// TIA Portal V20 export
// export: Created 2025-12-01T14:57:15.1286003Z, ExportSetting None, DisplayName Totally Integrated Automation Portal, DisplayVersion V20 Update 3, DisplayName TIA Portal Openness, DisplayVersion V20 Update 3, DisplayName TIA Portal Version Control Interface, DisplayVersion V20 Update 3, DisplayName STEP 7 Professional, DisplayVersion V20 Update 3, DisplayName STEP 7 Safety, DisplayVersion V20 Update 2, DisplayName WinCC Basic/Comfort/Advanced, DisplayVersion V20 Update 3, DisplayName WinCC Professional, DisplayVersion V20 Update 3, DisplayName WinCC Unified, DisplayVersion V20 Update 3
FUNCTION_BLOCK "FB900_CONTROL_ZONA"   // FB900, LAD
{ S7_Optimized_Access := 'FALSE' }
AUTHOR : ESTANDAR
NAME : 20160526
VERSION : 3.4
// stored: AutoNumber false, SetENOAutomatically false
   VAR_INPUT
      NumZonaUP : UInt;
      NumZona : UInt;
      MAR_FinReset_DW : Bool;   // FIN RESET MESAS INTEGRANTES CBOX
      CONF_Reset_Manual : Bool;   // Reset Manual
      INP_Sel_OffLine : Bool;
      INP_Sel_Main : Bool;
      INP_Pul_Marcha : Bool;   // Pulsador Manual Zona
      INP_Pul_Paro : Bool;   // Pulsador Paro Zona
      INP_Pul_Rearme : Bool;   // Pulsador Test Luces CCPIF
      INP_Pul_TLuces : Bool;   // Pulsador Test Luces Zona
      INP_Sel_Automat : Bool;   // Selector Automatico Zona
      INP_Sel_Manual : Bool;   // Selector Automatico Zona
   END_VAR
   VAR_OUTPUT
      L_Verde : Bool;   // Piloto Marcha
      L_Rojo : Bool;   // Piloto Error
      L_Naranja : Bool;
      Sirena : Bool;
   END_VAR
   VAR
      Toff_Rearme { ExternalAccessible := 'False'; ExternalVisible := 'False'; ExternalWritable := 'False'} : TOF_TIME;
      TIM_RetardoMarcha { S7_SetPoint := 'True'} : TON_TIME;
      Valor_Cuenta_Reset : UDInt;   // No comment
      Modo_Zona_E0 : Bool;   // Gragcet Modo
      Modo_Zona_E1 : Bool;   // Gragcet Modo
      Modo_Zona_E2 : Bool;   // Gragcet Modo
      Modo_Zona_E3 : Bool;   // Gragcet Modo
      Modo_Zona_E4 : Bool;   // Gragcet Modo
      Modo_Zona_E5 : Bool;   // Gragcet Modo
      S_Paro_Zona : Bool;   // Sel_Paro
      S_Marcha_Zona : Bool;   // Sel_Marcha
      Auto_Zona_E0 : Bool;   // Grafcet Auto
      Auto_Zona_E1 : Bool;   // Grafcet Auto
      Auto_Zona_E2 : Bool;   // Grafcet Auto
      Auto_Zona_E3 : Bool;   // Grafcet Auto
      Auto_Zona_E4 : Bool;   // Grafcet Auto
      Auto_Zona_E5 : Bool;   // Grafcet Auto
      Reset_Zona_E0 : Bool;   // Grafcet Reset
      Reset_Zona_E1 : Bool;   // Grafcet Reset
      Reset_Zona_E2 : Bool;   // Grafcet Reset
      Reset_Zona_E3 : Bool;   // Grafcet Reset
      Reset_Zona_E4 : Bool;   // Grafcet Reset
      Reset_Zona_E5 : Bool;   // Grafcet Reset
      Reset_Zona_E6 : Bool;   // Grafcet Reset
      Reset_Zona_E7 : Bool;   // Grafcet Reset
      Mem_PulMarcha_Zona : Bool;   // Mem_Auxiliar
      Mem_Error_Zona : Bool;   // Mem_Auxiliar
      Mem_Aviso_Error_Zona : Bool;   // Mem_Auxiliar
      Mem_Parar_Zona : Bool;   // Mem_Auxiliar
      Mem_Reseteo_Zona : Bool;   // Mem_Auxiliar
      Mem_PulParo_Zona : Bool;   // Mem_Auxiliar
      Mem_Fin_Zona : Bool;   // Mem_Auxiliar
      Mem_Fin_Reset_Zona : Bool;   // Mem_Auxiliar
      Mem_FP_Rearme : Bool;   // Mem_Auxiliar
      Mem_Free2 : Bool;   // Mem_Auxiliar
      MemoriaSirena : Bool;
      Cuenta_Reset_OK : Bool;   // No comment
   END_VAR
   VAR_TEMP
      Zona : "UDT_EstadoZonaDispositivo";   // Estado de la Zona
      ZonaUP : "UDT_EstadoZonaDispositivo";   // Estado de la Zona UP
      Tmp_Cod_Error_DInt : DInt;   // No comment
      NumDispo : UInt;
      NumDispoUP : UInt;
      Cero : Byte;
      ValorReturn : Int;
      FlancoPulsadorMarcha : Bool;   // FP Pulsador Marcha
      FlancoPulsadorParo : Bool;   // FP. Pulsador Paro
      FlancoReset : Bool;   // FP. Reset
   END_VAR
   VAR_TEMP   // added for the SCL form of the ladder/FBD networks
      _w1 : Bool;
      _w2 : Bool;
   END_VAR
BEGIN

NETWORK
TITLE = Inicio
// ---------------------------------------------------------------------
// --- Paso 1 : Inicio de Variables

      L     #NumZona;  // - Numero de Zona
      T     #NumDispo;

      L     #NumZonaUP;  // - Numero de Zona UP
      T     #NumDispoUP;


// ---------------------------------------------------------------------
// --- Paso 2 : Leer datos del DB de Zona

      CALL  BLKMOV
      ( SRCBLK  := "DB901_Estado_Zonas".EstadoZona[#NumDispo],
        RET_VAL := #ValorReturn,
        DSTBLK  := #Zona
      );


// ---------------------------------------------------------------------
// --- Paso 3 : Leer datos del DB de Zona UP

      L     #NumDispo;  // - Comprobar Si tiene Zona UP
      L     #NumDispoUP;
      <>I;
      JC    S_UP;

      L     0;  // Inicializo
      T     #Cero;
      CALL  FILL
      ( BVAL    := #Cero,
        RET_VAL := #ValorReturn,
        BLK     := #ZonaUP
      );

      A     "ON";
      S     #ZonaUP.Estado.Marcha_CBx;
      S     #ZonaUP.Estado.Automatico_CBx;
      S     #ZonaUP.Pulsador.MemoriaPulsadorParo;

      JU    FP_5;

S_UP: NOP   0;

      CALL  BLKMOV
      ( SRCBLK  := "DB901_Estado_Zonas".EstadoZona[#NumDispoUP],
        RET_VAL := #ValorReturn,
        DSTBLK  := #ZonaUP
      );

      JU    FP_5;


FP_5: NOP   0;




REGION Network 2: Calcular Codigo de Error -- Emergencia
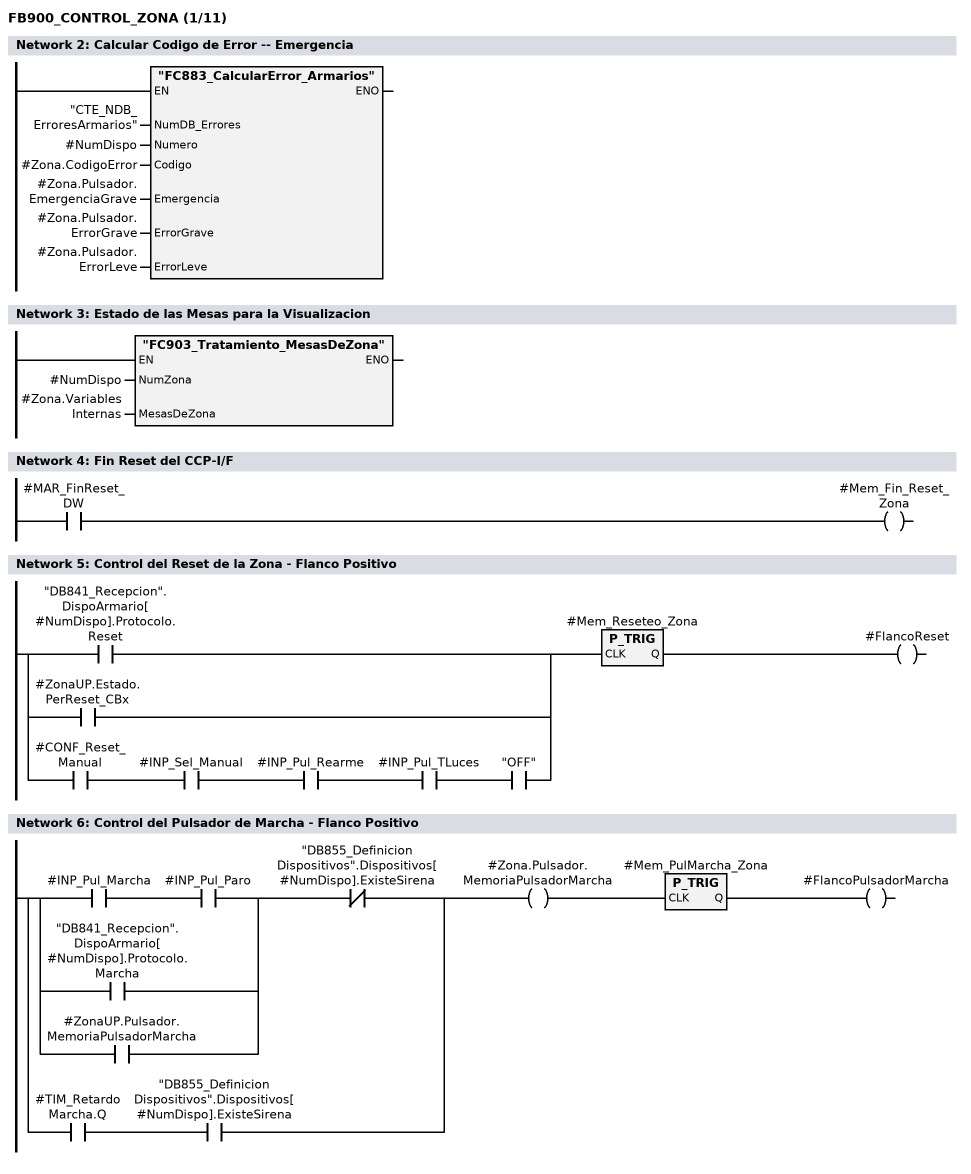
   RUNG wire#powerrail
      "FC883_CalcularError_Armarios"(NumDB_Errores := "CTE_NDB_ErroresArmarios", Numero := #NumDispo, Codigo := #Zona.CodigoError, Emergencia := #Zona.Pulsador.EmergenciaGrave, ErrorGrave := #Zona.Pulsador.ErrorGrave, ErrorLeve := #Zona.Pulsador.ErrorLeve)
   END_RUNG
   // the same network as SCL:
   "FC883_CalcularError_Armarios"(NumDB_Errores := "CTE_NDB_ErroresArmarios",
                           Numero := #NumDispo,
                           Codigo := #Zona.CodigoError,
                           Emergencia := #Zona.Pulsador.EmergenciaGrave,
                           ErrorGrave := #Zona.Pulsador.ErrorGrave,
                           ErrorLeve := #Zona.Pulsador.ErrorLeve);
END_REGION

REGION Network 3: Estado de las Mesas para la Visualizacion
   RUNG wire#powerrail
      "FC903_Tratamiento_MesasDeZona"(NumZona := #NumDispo, MesasDeZona := #Zona.VariablesInternas)
   END_RUNG
   // the same network as SCL:
   "FC903_Tratamiento_MesasDeZona"(NumZona := #NumDispo, MesasDeZona := #Zona.VariablesInternas);
END_REGION

REGION Network 4: Fin Reset del CCP-I/F
   RUNG wire#powerrail
      Contact( #MAR_FinReset_DW )
      Coil( #Mem_Fin_Reset_Zona )
   END_RUNG
   // the same network as SCL:
   #Mem_Fin_Reset_Zona := #MAR_FinReset_DW;
END_REGION

REGION Network 5: Control del Reset de la Zona - Flanco Positivo
   RUNG wire#powerrail
      Contact( "DB841_Recepcion".DispoArmario[#NumDispo].Protocolo.Reset )
      wire#w1
      P_Trig( #Mem_Reseteo_Zona )
      Coil( #FlancoReset )
   END_RUNG
   RUNG wire#powerrail
      Contact( #ZonaUP.Estado.PerReset_CBx )
   END_RUNG wire#w1
   RUNG wire#powerrail
      Contact( #CONF_Reset_Manual )
      Contact( #INP_Sel_Manual )
      Contact( #INP_Pul_Rearme )
      Contact( #INP_Pul_TLuces )
      Contact( "OFF" )
   END_RUNG wire#w1
   // the same network as SCL:
   #_w1 := "DB841_Recepcion".DispoArmario[#NumDispo].Protocolo.Reset OR #ZonaUP.Estado.PerReset_CBx OR (#CONF_Reset_Manual AND #INP_Sel_Manual AND #INP_Pul_Rearme AND #INP_Pul_TLuces AND "OFF");
   #_w2 := #_w1 AND NOT #Mem_Reseteo_Zona;   // rising edge
   #Mem_Reseteo_Zona := #_w1;
   #FlancoReset := #_w2;
END_REGION

REGION Network 6: Control del Pulsador de Marcha - Flanco Positivo
   RUNG wire#powerrail
      Contact( #INP_Pul_Marcha )
      Contact( #INP_Pul_Paro )
      wire#w1
      I_Contact( "DB855_DefinicionDispositivos".Dispositivos[#NumDispo].ExisteSirena )
      wire#w2
      Coil( #Zona.Pulsador.MemoriaPulsadorMarcha )
      P_Trig( #Mem_PulMarcha_Zona )
      Coil( #FlancoPulsadorMarcha )
   END_RUNG
   RUNG wire#powerrail
      Contact( "DB841_Recepcion".DispoArmario[#NumDispo].Protocolo.Marcha )
   END_RUNG wire#w1
   RUNG wire#powerrail
      Contact( #ZonaUP.Pulsador.MemoriaPulsadorMarcha )
   END_RUNG wire#w1
   RUNG wire#powerrail
      Contact( #TIM_RetardoMarcha.Q )
      Contact( "DB855_DefinicionDispositivos".Dispositivos[#NumDispo].ExisteSirena )
   END_RUNG wire#w2
   // the same network as SCL:
   #Zona.Pulsador.MemoriaPulsadorMarcha := (((#INP_Pul_Marcha AND #INP_Pul_Paro) OR "DB841_Recepcion".DispoArmario[#NumDispo].Protocolo.Marcha OR #ZonaUP.Pulsador.MemoriaPulsadorMarcha) AND NOT "DB855_DefinicionDispositivos".Dispositivos[#NumDispo].ExisteSirena) OR (#TIM_RetardoMarcha.Q AND "DB855_DefinicionDispositivos".Dispositivos[#NumDispo].ExisteSirena);
   #_w1 := #Zona.Pulsador.MemoriaPulsadorMarcha AND NOT #Mem_PulMarcha_Zona;   // rising edge
   #Mem_PulMarcha_Zona := #Zona.Pulsador.MemoriaPulsadorMarcha;
   #FlancoPulsadorMarcha := #_w1;
END_REGION

REGION Network 7: Control del Pulsador de Paro - Flanco Positivo
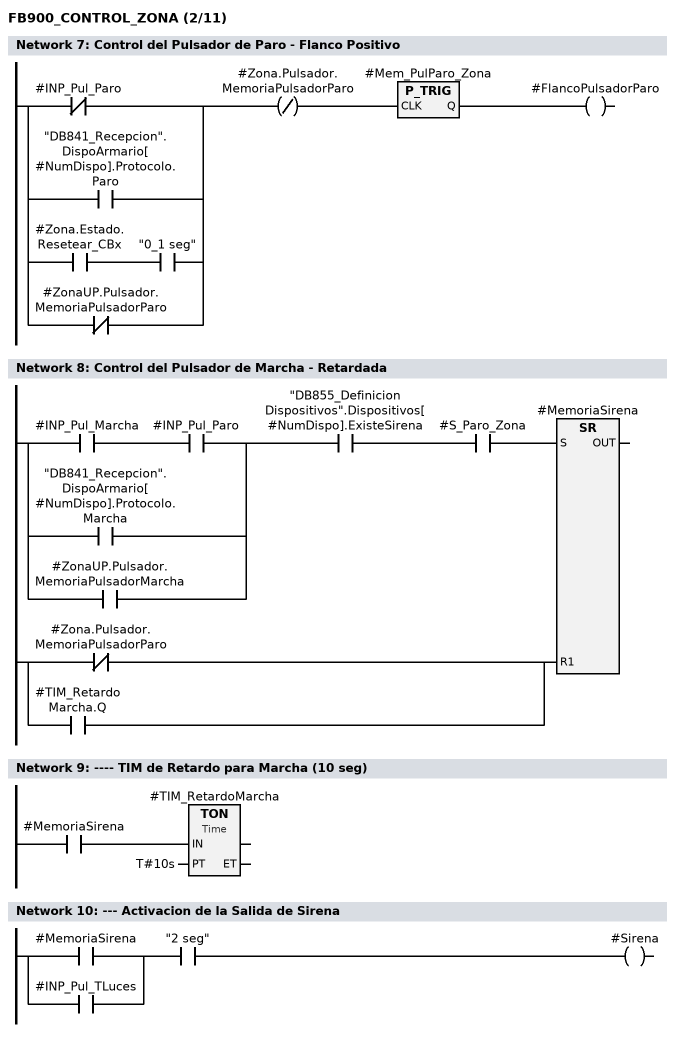
   RUNG wire#powerrail
      I_Contact( #INP_Pul_Paro )
      wire#w1
      I_Coil( #Zona.Pulsador.MemoriaPulsadorParo )
      P_Trig( #Mem_PulParo_Zona )
      Coil( #FlancoPulsadorParo )
   END_RUNG
   RUNG wire#powerrail
      Contact( "DB841_Recepcion".DispoArmario[#NumDispo].Protocolo.Paro )
   END_RUNG wire#w1
   RUNG wire#powerrail
      Contact( #Zona.Estado.Resetear_CBx )
      Contact( "0_1 seg" )
   END_RUNG wire#w1
   RUNG wire#powerrail
      I_Contact( #ZonaUP.Pulsador.MemoriaPulsadorParo )
   END_RUNG wire#w1
   // the same network as SCL:
   #_w1 := NOT #INP_Pul_Paro OR "DB841_Recepcion".DispoArmario[#NumDispo].Protocolo.Paro OR (#Zona.Estado.Resetear_CBx AND "0_1 seg") OR NOT #ZonaUP.Pulsador.MemoriaPulsadorParo;
   #Zona.Pulsador.MemoriaPulsadorParo := NOT #_w1;
   #_w2 := #_w1 AND NOT #Mem_PulParo_Zona;   // rising edge
   #Mem_PulParo_Zona := #_w1;
   #FlancoPulsadorParo := #_w2;
END_REGION

REGION Network 8: Control del Pulsador de Marcha - Retardada
   RUNG wire#powerrail
      Contact( #INP_Pul_Marcha )
      Contact( #INP_Pul_Paro )
      wire#w1
      Contact( "DB855_DefinicionDispositivos".Dispositivos[#NumDispo].ExisteSirena )
      Contact( #S_Paro_Zona )
      S_SR(operand := #MemoriaSirena, r1 := wire#w2)
   END_RUNG
   RUNG wire#powerrail
      Contact( "DB841_Recepcion".DispoArmario[#NumDispo].Protocolo.Marcha )
   END_RUNG wire#w1
   RUNG wire#powerrail
      Contact( #ZonaUP.Pulsador.MemoriaPulsadorMarcha )
   END_RUNG wire#w1
   RUNG wire#powerrail
      I_Contact( #Zona.Pulsador.MemoriaPulsadorParo )
   END_RUNG wire#w2
   RUNG wire#powerrail
      Contact( #TIM_RetardoMarcha.Q )
   END_RUNG wire#w2
   // the same network as SCL:
   IF ((#INP_Pul_Marcha AND #INP_Pul_Paro) OR "DB841_Recepcion".DispoArmario[#NumDispo].Protocolo.Marcha OR #ZonaUP.Pulsador.MemoriaPulsadorMarcha) AND "DB855_DefinicionDispositivos".Dispositivos[#NumDispo].ExisteSirena AND #S_Paro_Zona THEN
       #MemoriaSirena := TRUE;   // SR flip-flop
   END_IF;
   IF NOT #Zona.Pulsador.MemoriaPulsadorParo OR #TIM_RetardoMarcha.Q THEN #MemoriaSirena := FALSE; END_IF;
END_REGION

REGION Network 9: ---- TIM de Retardo para Marcha (10 seg)
   RUNG wire#powerrail
      Contact( #MemoriaSirena )
      { S7_Templates := "time_type := Time" } #TIM_RetardoMarcha.TON(pt := T#10s, et =>)
   END_RUNG
   // the same network as SCL:
   #TIM_RetardoMarcha(IN := #MemoriaSirena, PT := T#10s);   // TON
END_REGION

REGION Network 10: --- Activacion de la Salida de Sirena
   RUNG wire#powerrail
      Contact( #MemoriaSirena )
      wire#w1
      Contact( "2 seg" )
      Coil( #Sirena )
   END_RUNG
   RUNG wire#powerrail
      Contact( #INP_Pul_TLuces )
   END_RUNG wire#w1
   // the same network as SCL:
   #Sirena := (#MemoriaSirena OR #INP_Pul_TLuces) AND "2 seg";
END_REGION

REGION Network 11: Sistema En Marcha de la Zona
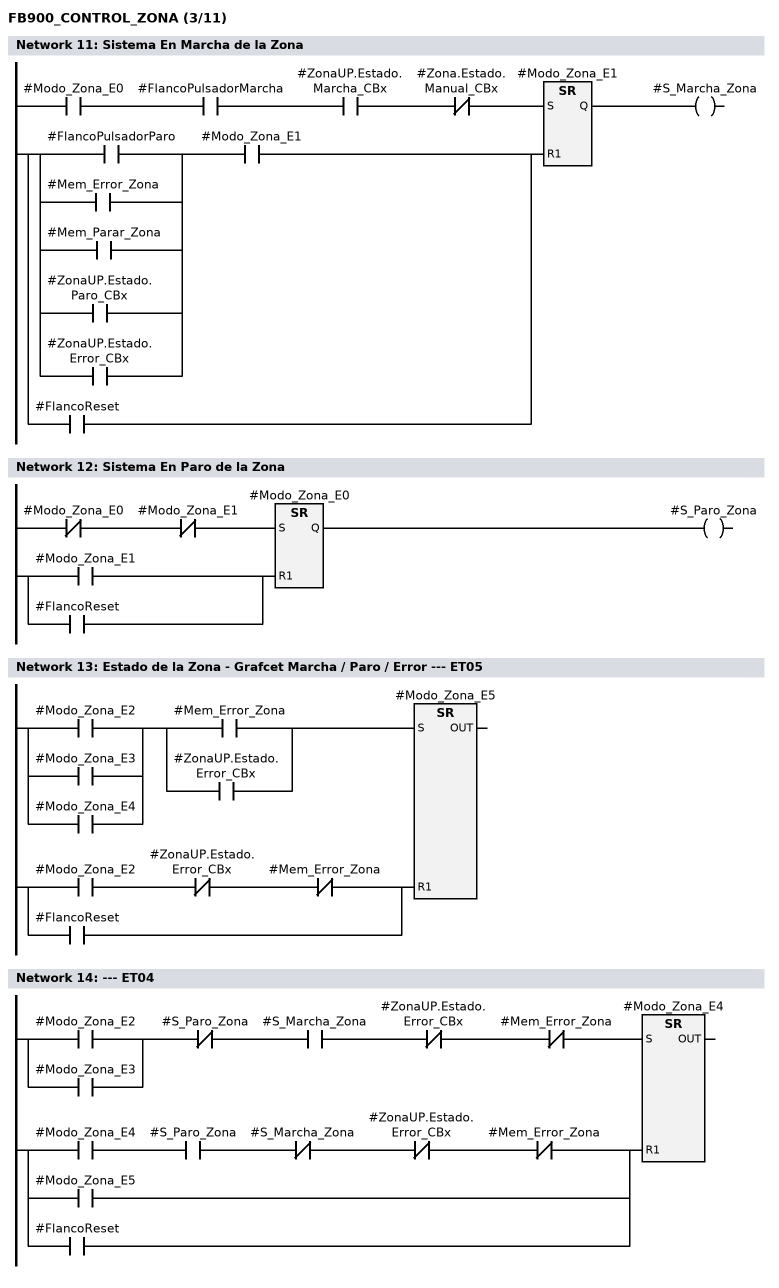
   RUNG wire#powerrail
      Contact( #Modo_Zona_E0 )
      Contact( #FlancoPulsadorMarcha )
      Contact( #ZonaUP.Estado.Marcha_CBx )
      I_Contact( #Zona.Estado.Manual_CBx )
      S_SR(operand := #Modo_Zona_E1, r1 := wire#w2)
      Coil( #S_Marcha_Zona )
   END_RUNG
   RUNG wire#powerrail
      Contact( #FlancoPulsadorParo )
      wire#w1
      Contact( #Modo_Zona_E1 )
   END_RUNG wire#w2
   RUNG wire#powerrail
      Contact( #Mem_Error_Zona )
   END_RUNG wire#w1
   RUNG wire#powerrail
      Contact( #Mem_Parar_Zona )
   END_RUNG wire#w1
   RUNG wire#powerrail
      Contact( #ZonaUP.Estado.Paro_CBx )
   END_RUNG wire#w1
   RUNG wire#powerrail
      Contact( #ZonaUP.Estado.Error_CBx )
   END_RUNG wire#w1
   RUNG wire#powerrail
      Contact( #FlancoReset )
   END_RUNG wire#w2
   // the same network as SCL:
   #_w1 := ((#FlancoPulsadorParo OR #Mem_Error_Zona OR #Mem_Parar_Zona OR #ZonaUP.Estado.Paro_CBx OR #ZonaUP.Estado.Error_CBx) AND #Modo_Zona_E1) OR #FlancoReset;
   IF #Modo_Zona_E0 AND #FlancoPulsadorMarcha AND #ZonaUP.Estado.Marcha_CBx AND NOT #Zona.Estado.Manual_CBx THEN
       #Modo_Zona_E1 := TRUE;   // SR flip-flop
   END_IF;
   IF #_w1 THEN #Modo_Zona_E1 := FALSE; END_IF;
   #S_Marcha_Zona := #Modo_Zona_E1;
END_REGION

REGION Network 12: Sistema En Paro de la Zona
   RUNG wire#powerrail
      I_Contact( #Modo_Zona_E0 )
      I_Contact( #Modo_Zona_E1 )
      S_SR(operand := #Modo_Zona_E0, r1 := wire#w1)
      Coil( #S_Paro_Zona )
   END_RUNG
   RUNG wire#powerrail
      Contact( #Modo_Zona_E1 )
   END_RUNG wire#w1
   RUNG wire#powerrail
      Contact( #FlancoReset )
   END_RUNG wire#w1
   // the same network as SCL:
   IF NOT #Modo_Zona_E0 AND NOT #Modo_Zona_E1 THEN
       #Modo_Zona_E0 := TRUE;   // SR flip-flop
   END_IF;
   IF #Modo_Zona_E1 OR #FlancoReset THEN #Modo_Zona_E0 := FALSE; END_IF;
   #S_Paro_Zona := #Modo_Zona_E0;
END_REGION

REGION Network 13: Estado de la Zona - Grafcet Marcha / Paro / Error --- ET05
   RUNG wire#powerrail
      Contact( #Modo_Zona_E2 )
      wire#w1
      Contact( #Mem_Error_Zona )
      wire#w2
      S_SR(operand := #Modo_Zona_E5, r1 := wire#w3)
   END_RUNG
   RUNG wire#powerrail
      Contact( #Modo_Zona_E3 )
   END_RUNG wire#w1
   RUNG wire#powerrail
      Contact( #Modo_Zona_E4 )
   END_RUNG wire#w1
   RUNG wire#w1
      Contact( #ZonaUP.Estado.Error_CBx )
   END_RUNG wire#w2
   RUNG wire#powerrail
      Contact( #Modo_Zona_E2 )
      I_Contact( #ZonaUP.Estado.Error_CBx )
      I_Contact( #Mem_Error_Zona )
   END_RUNG wire#w3
   RUNG wire#powerrail
      Contact( #FlancoReset )
   END_RUNG wire#w3
   // the same network as SCL:
   IF (#Modo_Zona_E2 OR #Modo_Zona_E3 OR #Modo_Zona_E4) AND (#Mem_Error_Zona OR #ZonaUP.Estado.Error_CBx) THEN
       #Modo_Zona_E5 := TRUE;   // SR flip-flop
   END_IF;
   IF (#Modo_Zona_E2 AND NOT #ZonaUP.Estado.Error_CBx AND NOT #Mem_Error_Zona) OR #FlancoReset THEN
       #Modo_Zona_E5 := FALSE;
   END_IF;
END_REGION

REGION Network 14: --- ET04
   RUNG wire#powerrail
      Contact( #Modo_Zona_E2 )
      wire#w1
      I_Contact( #S_Paro_Zona )
      Contact( #S_Marcha_Zona )
      I_Contact( #ZonaUP.Estado.Error_CBx )
      I_Contact( #Mem_Error_Zona )
      S_SR(operand := #Modo_Zona_E4, r1 := wire#w2)
   END_RUNG
   RUNG wire#powerrail
      Contact( #Modo_Zona_E3 )
   END_RUNG wire#w1
   RUNG wire#powerrail
      Contact( #Modo_Zona_E4 )
      Contact( #S_Paro_Zona )
      I_Contact( #S_Marcha_Zona )
      I_Contact( #ZonaUP.Estado.Error_CBx )
      I_Contact( #Mem_Error_Zona )
   END_RUNG wire#w2
   RUNG wire#powerrail
      Contact( #Modo_Zona_E5 )
   END_RUNG wire#w2
   RUNG wire#powerrail
      Contact( #FlancoReset )
   END_RUNG wire#w2
   // the same network as SCL:
   #_w1 := (#Modo_Zona_E4 AND #S_Paro_Zona AND NOT #S_Marcha_Zona AND NOT #ZonaUP.Estado.Error_CBx AND NOT #Mem_Error_Zona) OR #Modo_Zona_E5 OR #FlancoReset;
   IF (#Modo_Zona_E2 OR #Modo_Zona_E3) AND NOT #S_Paro_Zona AND #S_Marcha_Zona AND NOT #ZonaUP.Estado.Error_CBx AND NOT #Mem_Error_Zona THEN
       #Modo_Zona_E4 := TRUE;   // SR flip-flop
   END_IF;
   IF #_w1 THEN #Modo_Zona_E4 := FALSE; END_IF;
END_REGION

REGION Network 15: --- ET03
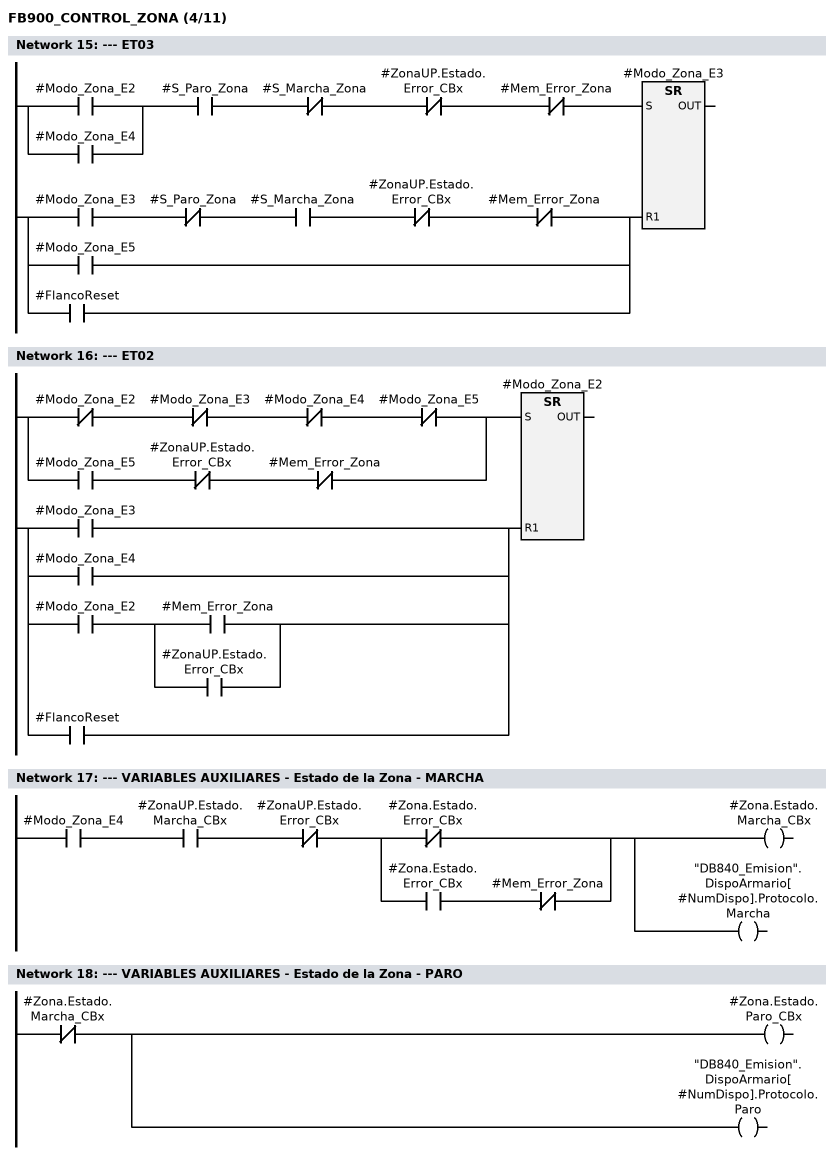
   RUNG wire#powerrail
      Contact( #Modo_Zona_E2 )
      wire#w1
      Contact( #S_Paro_Zona )
      I_Contact( #S_Marcha_Zona )
      I_Contact( #ZonaUP.Estado.Error_CBx )
      I_Contact( #Mem_Error_Zona )
      S_SR(operand := #Modo_Zona_E3, r1 := wire#w2)
   END_RUNG
   RUNG wire#powerrail
      Contact( #Modo_Zona_E4 )
   END_RUNG wire#w1
   RUNG wire#powerrail
      Contact( #Modo_Zona_E3 )
      I_Contact( #S_Paro_Zona )
      Contact( #S_Marcha_Zona )
      I_Contact( #ZonaUP.Estado.Error_CBx )
      I_Contact( #Mem_Error_Zona )
   END_RUNG wire#w2
   RUNG wire#powerrail
      Contact( #Modo_Zona_E5 )
   END_RUNG wire#w2
   RUNG wire#powerrail
      Contact( #FlancoReset )
   END_RUNG wire#w2
   // the same network as SCL:
   #_w1 := (#Modo_Zona_E3 AND NOT #S_Paro_Zona AND #S_Marcha_Zona AND NOT #ZonaUP.Estado.Error_CBx AND NOT #Mem_Error_Zona) OR #Modo_Zona_E5 OR #FlancoReset;
   IF (#Modo_Zona_E2 OR #Modo_Zona_E4) AND #S_Paro_Zona AND NOT #S_Marcha_Zona AND NOT #ZonaUP.Estado.Error_CBx AND NOT #Mem_Error_Zona THEN
       #Modo_Zona_E3 := TRUE;   // SR flip-flop
   END_IF;
   IF #_w1 THEN #Modo_Zona_E3 := FALSE; END_IF;
END_REGION

REGION Network 16: --- ET02
   RUNG wire#powerrail
      I_Contact( #Modo_Zona_E2 )
      I_Contact( #Modo_Zona_E3 )
      I_Contact( #Modo_Zona_E4 )
      I_Contact( #Modo_Zona_E5 )
      wire#w1
      S_SR(operand := #Modo_Zona_E2, r1 := wire#w3)
   END_RUNG
   RUNG wire#powerrail
      Contact( #Modo_Zona_E5 )
      I_Contact( #ZonaUP.Estado.Error_CBx )
      I_Contact( #Mem_Error_Zona )
   END_RUNG wire#w1
   RUNG wire#powerrail
      Contact( #Modo_Zona_E3 )
   END_RUNG wire#w3
   RUNG wire#powerrail
      Contact( #Modo_Zona_E4 )
   END_RUNG wire#w3
   RUNG wire#powerrail
      Contact( #Modo_Zona_E2 )
      wire#w2
      Contact( #Mem_Error_Zona )
   END_RUNG wire#w3
   RUNG wire#w2
      Contact( #ZonaUP.Estado.Error_CBx )
   END_RUNG wire#w3
   RUNG wire#powerrail
      Contact( #FlancoReset )
   END_RUNG wire#w3
   // the same network as SCL:
   #_w1 := #Modo_Zona_E3 OR #Modo_Zona_E4 OR (#Modo_Zona_E2 AND (#Mem_Error_Zona OR #ZonaUP.Estado.Error_CBx)) OR #FlancoReset;
   IF (NOT #Modo_Zona_E2 AND NOT #Modo_Zona_E3 AND NOT #Modo_Zona_E4 AND NOT #Modo_Zona_E5) OR (#Modo_Zona_E5 AND NOT #ZonaUP.Estado.Error_CBx AND NOT #Mem_Error_Zona) THEN
       #Modo_Zona_E2 := TRUE;   // SR flip-flop
   END_IF;
   IF #_w1 THEN #Modo_Zona_E2 := FALSE; END_IF;
END_REGION

REGION Network 17: --- VARIABLES AUXILIARES - Estado de la Zona - MARCHA
   RUNG wire#powerrail
      Contact( #Modo_Zona_E4 )
      Contact( #ZonaUP.Estado.Marcha_CBx )
      I_Contact( #ZonaUP.Estado.Error_CBx )
      wire#w1
      I_Contact( #Zona.Estado.Error_CBx )
      wire#w2
      Coil( #Zona.Estado.Marcha_CBx )
   END_RUNG
   RUNG wire#w1
      Contact( #Zona.Estado.Error_CBx )
      I_Contact( #Mem_Error_Zona )
   END_RUNG wire#w2
   RUNG wire#w2
      Coil( "DB840_Emision".DispoArmario[#NumDispo].Protocolo.Marcha )
   END_RUNG
   // the same network as SCL:
   #Zona.Estado.Marcha_CBx := #Modo_Zona_E4 AND #ZonaUP.Estado.Marcha_CBx AND NOT #ZonaUP.Estado.Error_CBx AND (NOT #Zona.Estado.Error_CBx OR (#Zona.Estado.Error_CBx AND NOT #Mem_Error_Zona));
   "DB840_Emision".DispoArmario[#NumDispo].Protocolo.Marcha := #Zona.Estado.Marcha_CBx;
END_REGION

REGION Network 18: --- VARIABLES AUXILIARES - Estado de la Zona - PARO
   RUNG wire#powerrail
      I_Contact( #Zona.Estado.Marcha_CBx )
      wire#w1
      Coil( #Zona.Estado.Paro_CBx )
   END_RUNG
   RUNG wire#w1
      Coil( "DB840_Emision".DispoArmario[#NumDispo].Protocolo.Paro )
   END_RUNG
   // the same network as SCL:
   #Zona.Estado.Paro_CBx := NOT #Zona.Estado.Marcha_CBx;
   "DB840_Emision".DispoArmario[#NumDispo].Protocolo.Paro := NOT #Zona.Estado.Marcha_CBx;
END_REGION

REGION Network 19: Estado de la Zona - Grafect Automatico / Manual / Remoto --- ET05 (DESAPERECE REMOTO)
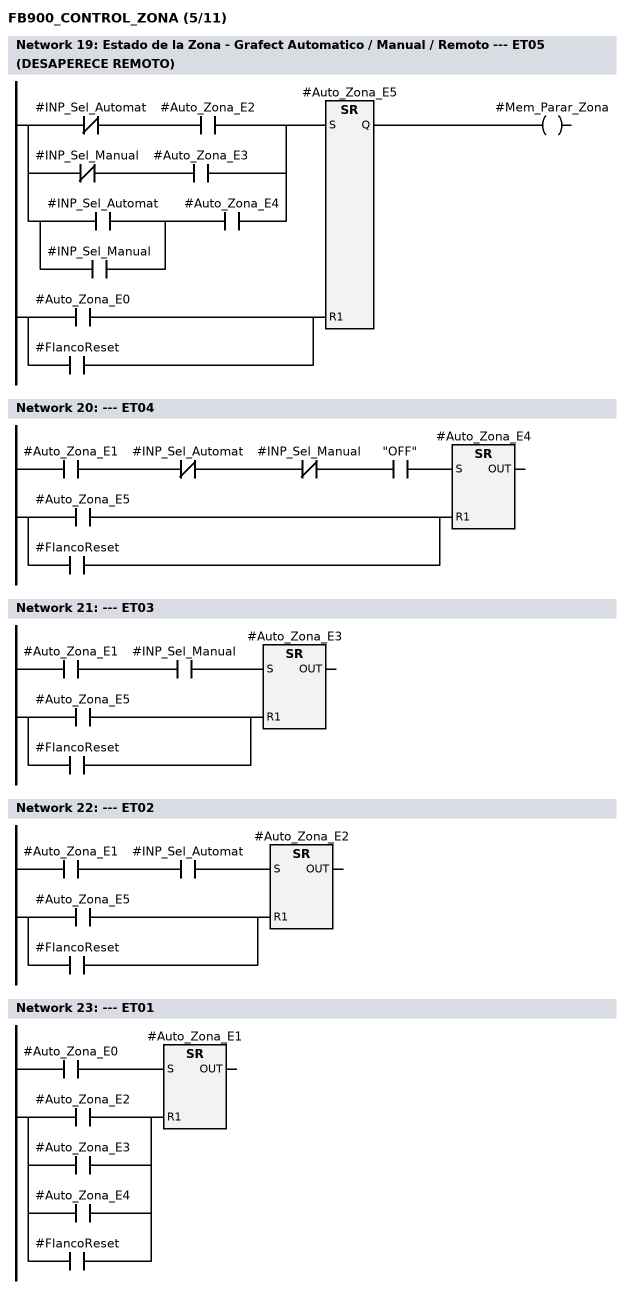
   RUNG wire#powerrail
      I_Contact( #INP_Sel_Automat )
      Contact( #Auto_Zona_E2 )
      wire#w1
      S_SR(operand := #Auto_Zona_E5, r1 := wire#w3)
      Coil( #Mem_Parar_Zona )
   END_RUNG
   RUNG wire#powerrail
      I_Contact( #INP_Sel_Manual )
      Contact( #Auto_Zona_E3 )
   END_RUNG wire#w1
   RUNG wire#powerrail
      Contact( #INP_Sel_Automat )
      wire#w2
      Contact( #Auto_Zona_E4 )
   END_RUNG wire#w1
   RUNG wire#powerrail
      Contact( #INP_Sel_Manual )
   END_RUNG wire#w2
   RUNG wire#powerrail
      Contact( #Auto_Zona_E0 )
   END_RUNG wire#w3
   RUNG wire#powerrail
      Contact( #FlancoReset )
   END_RUNG wire#w3
   // the same network as SCL:
   IF (NOT #INP_Sel_Automat AND #Auto_Zona_E2) OR (NOT #INP_Sel_Manual AND #Auto_Zona_E3) OR ((#INP_Sel_Automat OR #INP_Sel_Manual) AND #Auto_Zona_E4) THEN
       #Auto_Zona_E5 := TRUE;   // SR flip-flop
   END_IF;
   IF #Auto_Zona_E0 OR #FlancoReset THEN #Auto_Zona_E5 := FALSE; END_IF;
   #Mem_Parar_Zona := #Auto_Zona_E5;
END_REGION

REGION Network 20: --- ET04
   RUNG wire#powerrail
      Contact( #Auto_Zona_E1 )
      I_Contact( #INP_Sel_Automat )
      I_Contact( #INP_Sel_Manual )
      Contact( "OFF" )
      S_SR(operand := #Auto_Zona_E4, r1 := wire#w1)
   END_RUNG
   RUNG wire#powerrail
      Contact( #Auto_Zona_E5 )
   END_RUNG wire#w1
   RUNG wire#powerrail
      Contact( #FlancoReset )
   END_RUNG wire#w1
   // the same network as SCL:
   IF #Auto_Zona_E1 AND NOT #INP_Sel_Automat AND NOT #INP_Sel_Manual AND "OFF" THEN
       #Auto_Zona_E4 := TRUE;   // SR flip-flop
   END_IF;
   IF #Auto_Zona_E5 OR #FlancoReset THEN #Auto_Zona_E4 := FALSE; END_IF;
END_REGION

REGION Network 21: --- ET03
   RUNG wire#powerrail
      Contact( #Auto_Zona_E1 )
      Contact( #INP_Sel_Manual )
      S_SR(operand := #Auto_Zona_E3, r1 := wire#w1)
   END_RUNG
   RUNG wire#powerrail
      Contact( #Auto_Zona_E5 )
   END_RUNG wire#w1
   RUNG wire#powerrail
      Contact( #FlancoReset )
   END_RUNG wire#w1
   // the same network as SCL:
   IF #Auto_Zona_E1 AND #INP_Sel_Manual THEN
       #Auto_Zona_E3 := TRUE;   // SR flip-flop
   END_IF;
   IF #Auto_Zona_E5 OR #FlancoReset THEN #Auto_Zona_E3 := FALSE; END_IF;
END_REGION

REGION Network 22: --- ET02
   RUNG wire#powerrail
      Contact( #Auto_Zona_E1 )
      Contact( #INP_Sel_Automat )
      S_SR(operand := #Auto_Zona_E2, r1 := wire#w1)
   END_RUNG
   RUNG wire#powerrail
      Contact( #Auto_Zona_E5 )
   END_RUNG wire#w1
   RUNG wire#powerrail
      Contact( #FlancoReset )
   END_RUNG wire#w1
   // the same network as SCL:
   IF #Auto_Zona_E1 AND #INP_Sel_Automat THEN
       #Auto_Zona_E2 := TRUE;   // SR flip-flop
   END_IF;
   IF #Auto_Zona_E5 OR #FlancoReset THEN #Auto_Zona_E2 := FALSE; END_IF;
END_REGION

REGION Network 23: --- ET01
   RUNG wire#powerrail
      Contact( #Auto_Zona_E0 )
      S_SR(operand := #Auto_Zona_E1, r1 := wire#w1)
   END_RUNG
   RUNG wire#powerrail
      Contact( #Auto_Zona_E2 )
   END_RUNG wire#w1
   RUNG wire#powerrail
      Contact( #Auto_Zona_E3 )
   END_RUNG wire#w1
   RUNG wire#powerrail
      Contact( #Auto_Zona_E4 )
   END_RUNG wire#w1
   RUNG wire#powerrail
      Contact( #FlancoReset )
   END_RUNG wire#w1
   // the same network as SCL:
   IF #Auto_Zona_E0 THEN
       #Auto_Zona_E1 := TRUE;   // SR flip-flop
   END_IF;
   IF #Auto_Zona_E2 OR #Auto_Zona_E3 OR #Auto_Zona_E4 OR #FlancoReset THEN #Auto_Zona_E1 := FALSE; END_IF;
END_REGION

REGION Network 24: --- ET00
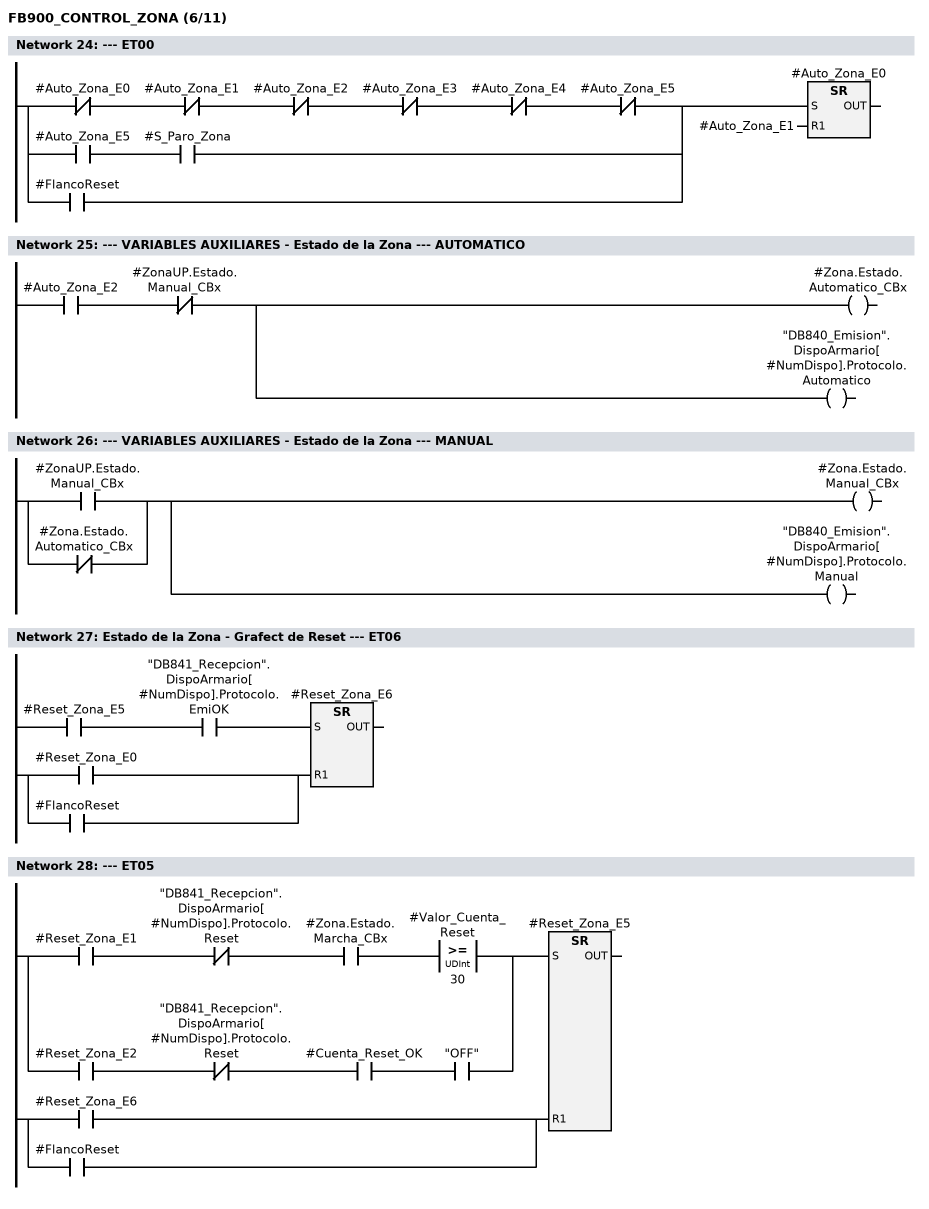
   RUNG wire#powerrail
      I_Contact( #Auto_Zona_E0 )
      I_Contact( #Auto_Zona_E1 )
      I_Contact( #Auto_Zona_E2 )
      I_Contact( #Auto_Zona_E3 )
      I_Contact( #Auto_Zona_E4 )
      I_Contact( #Auto_Zona_E5 )
      wire#w1
      S_SR(operand := #Auto_Zona_E0, r1 := #Auto_Zona_E1)
   END_RUNG
   RUNG wire#powerrail
      Contact( #Auto_Zona_E5 )
      Contact( #S_Paro_Zona )
   END_RUNG wire#w1
   RUNG wire#powerrail
      Contact( #FlancoReset )
   END_RUNG wire#w1
   // the same network as SCL:
   IF (NOT #Auto_Zona_E0 AND NOT #Auto_Zona_E1 AND NOT #Auto_Zona_E2 AND NOT #Auto_Zona_E3 AND NOT #Auto_Zona_E4 AND NOT #Auto_Zona_E5) OR (#Auto_Zona_E5 AND #S_Paro_Zona) OR #FlancoReset THEN
       #Auto_Zona_E0 := TRUE;   // SR flip-flop
   END_IF;
   IF #Auto_Zona_E1 THEN #Auto_Zona_E0 := FALSE; END_IF;
END_REGION

REGION Network 25: --- VARIABLES AUXILIARES - Estado de la Zona --- AUTOMATICO
   RUNG wire#powerrail
      Contact( #Auto_Zona_E2 )
      I_Contact( #ZonaUP.Estado.Manual_CBx )
      wire#w1
      Coil( #Zona.Estado.Automatico_CBx )
   END_RUNG
   RUNG wire#w1
      Coil( "DB840_Emision".DispoArmario[#NumDispo].Protocolo.Automatico )
   END_RUNG
   // the same network as SCL:
   #Zona.Estado.Automatico_CBx := #Auto_Zona_E2 AND NOT #ZonaUP.Estado.Manual_CBx;
   "DB840_Emision".DispoArmario[#NumDispo].Protocolo.Automatico := #Zona.Estado.Automatico_CBx;
END_REGION

REGION Network 26: --- VARIABLES AUXILIARES - Estado de la Zona --- MANUAL
   RUNG wire#powerrail
      Contact( #ZonaUP.Estado.Manual_CBx )
      wire#w1
      Coil( #Zona.Estado.Manual_CBx )
   END_RUNG
   RUNG wire#powerrail
      I_Contact( #Zona.Estado.Automatico_CBx )
   END_RUNG wire#w1
   RUNG wire#w1
      Coil( "DB840_Emision".DispoArmario[#NumDispo].Protocolo.Manual )
   END_RUNG
   // the same network as SCL:
   #Zona.Estado.Manual_CBx := #ZonaUP.Estado.Manual_CBx OR NOT #Zona.Estado.Automatico_CBx;
   "DB840_Emision".DispoArmario[#NumDispo].Protocolo.Manual := #Zona.Estado.Manual_CBx;
END_REGION

REGION Network 27: Estado de la Zona - Grafect de Reset --- ET06
   RUNG wire#powerrail
      Contact( #Reset_Zona_E5 )
      Contact( "DB841_Recepcion".DispoArmario[#NumDispo].Protocolo.EmiOK )
      S_SR(operand := #Reset_Zona_E6, r1 := wire#w1)
   END_RUNG
   RUNG wire#powerrail
      Contact( #Reset_Zona_E0 )
   END_RUNG wire#w1
   RUNG wire#powerrail
      Contact( #FlancoReset )
   END_RUNG wire#w1
   // the same network as SCL:
   IF #Reset_Zona_E5 AND "DB841_Recepcion".DispoArmario[#NumDispo].Protocolo.EmiOK THEN
       #Reset_Zona_E6 := TRUE;   // SR flip-flop
   END_IF;
   IF #Reset_Zona_E0 OR #FlancoReset THEN #Reset_Zona_E6 := FALSE; END_IF;
END_REGION

REGION Network 28: --- ET05
   RUNG wire#powerrail
      Contact( #Reset_Zona_E1 )
      I_Contact( "DB841_Recepcion".DispoArmario[#NumDispo].Protocolo.Reset )
      Contact( #Zona.Estado.Marcha_CBx )
      { S7_Templates := "SrcType := UDInt" } GE_Contact(in1 := #Valor_Cuenta_Reset, in2 := 30)
      wire#w1
      S_SR(operand := #Reset_Zona_E5, r1 := wire#w2)
   END_RUNG
   RUNG wire#powerrail
      Contact( #Reset_Zona_E2 )
      I_Contact( "DB841_Recepcion".DispoArmario[#NumDispo].Protocolo.Reset )
      Contact( #Cuenta_Reset_OK )
      Contact( "OFF" )
   END_RUNG wire#w1
   RUNG wire#powerrail
      Contact( #Reset_Zona_E6 )
   END_RUNG wire#w2
   RUNG wire#powerrail
      Contact( #FlancoReset )
   END_RUNG wire#w2
   // the same network as SCL:
   IF (#Reset_Zona_E1 AND NOT "DB841_Recepcion".DispoArmario[#NumDispo].Protocolo.Reset AND #Zona.Estado.Marcha_CBx AND (#Valor_Cuenta_Reset >= 30)) OR (#Reset_Zona_E2 AND NOT "DB841_Recepcion".DispoArmario[#NumDispo].Protocolo.Reset AND #Cuenta_Reset_OK AND "OFF") THEN
       #Reset_Zona_E5 := TRUE;   // SR flip-flop
   END_IF;
   IF #Reset_Zona_E6 OR #FlancoReset THEN #Reset_Zona_E5 := FALSE; END_IF;
END_REGION

REGION Network 29: --- ET04
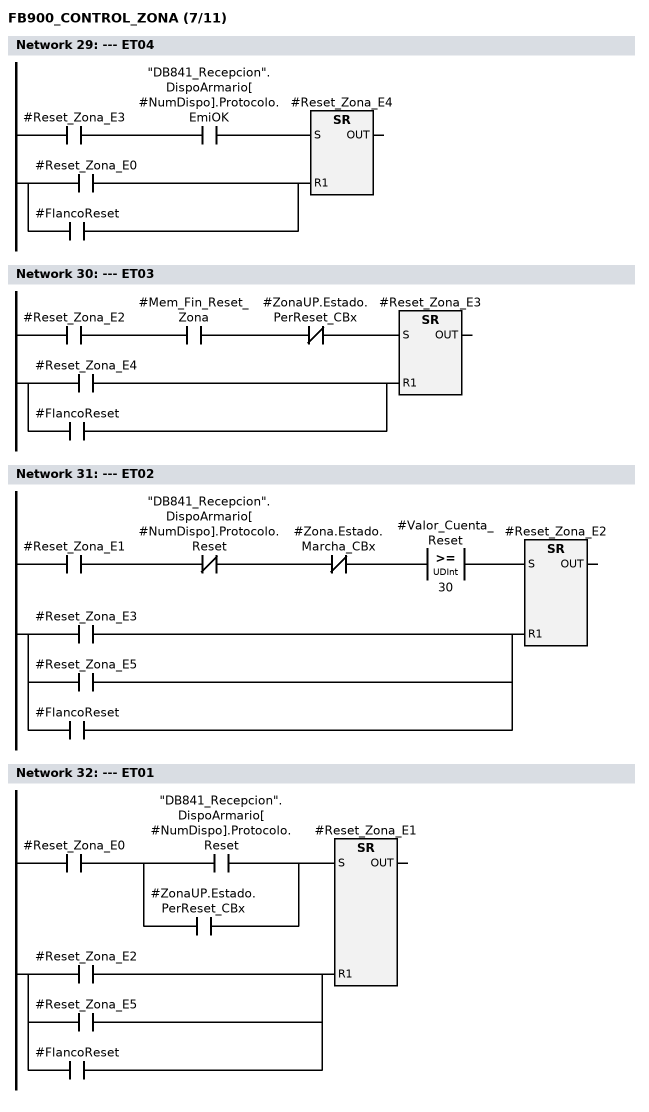
   RUNG wire#powerrail
      Contact( #Reset_Zona_E3 )
      Contact( "DB841_Recepcion".DispoArmario[#NumDispo].Protocolo.EmiOK )
      S_SR(operand := #Reset_Zona_E4, r1 := wire#w1)
   END_RUNG
   RUNG wire#powerrail
      Contact( #Reset_Zona_E0 )
   END_RUNG wire#w1
   RUNG wire#powerrail
      Contact( #FlancoReset )
   END_RUNG wire#w1
   // the same network as SCL:
   IF #Reset_Zona_E3 AND "DB841_Recepcion".DispoArmario[#NumDispo].Protocolo.EmiOK THEN
       #Reset_Zona_E4 := TRUE;   // SR flip-flop
   END_IF;
   IF #Reset_Zona_E0 OR #FlancoReset THEN #Reset_Zona_E4 := FALSE; END_IF;
END_REGION

REGION Network 30: --- ET03
   RUNG wire#powerrail
      Contact( #Reset_Zona_E2 )
      Contact( #Mem_Fin_Reset_Zona )
      I_Contact( #ZonaUP.Estado.PerReset_CBx )
      S_SR(operand := #Reset_Zona_E3, r1 := wire#w1)
   END_RUNG
   RUNG wire#powerrail
      Contact( #Reset_Zona_E4 )
   END_RUNG wire#w1
   RUNG wire#powerrail
      Contact( #FlancoReset )
   END_RUNG wire#w1
   // the same network as SCL:
   IF #Reset_Zona_E2 AND #Mem_Fin_Reset_Zona AND NOT #ZonaUP.Estado.PerReset_CBx THEN
       #Reset_Zona_E3 := TRUE;   // SR flip-flop
   END_IF;
   IF #Reset_Zona_E4 OR #FlancoReset THEN #Reset_Zona_E3 := FALSE; END_IF;
END_REGION

REGION Network 31: --- ET02
   RUNG wire#powerrail
      Contact( #Reset_Zona_E1 )
      I_Contact( "DB841_Recepcion".DispoArmario[#NumDispo].Protocolo.Reset )
      I_Contact( #Zona.Estado.Marcha_CBx )
      { S7_Templates := "SrcType := UDInt" } GE_Contact(in1 := #Valor_Cuenta_Reset, in2 := 30)
      S_SR(operand := #Reset_Zona_E2, r1 := wire#w1)
   END_RUNG
   RUNG wire#powerrail
      Contact( #Reset_Zona_E3 )
   END_RUNG wire#w1
   RUNG wire#powerrail
      Contact( #Reset_Zona_E5 )
   END_RUNG wire#w1
   RUNG wire#powerrail
      Contact( #FlancoReset )
   END_RUNG wire#w1
   // the same network as SCL:
   IF #Reset_Zona_E1 AND NOT "DB841_Recepcion".DispoArmario[#NumDispo].Protocolo.Reset AND NOT #Zona.Estado.Marcha_CBx AND (#Valor_Cuenta_Reset >= 30) THEN
       #Reset_Zona_E2 := TRUE;   // SR flip-flop
   END_IF;
   IF #Reset_Zona_E3 OR #Reset_Zona_E5 OR #FlancoReset THEN #Reset_Zona_E2 := FALSE; END_IF;
END_REGION

REGION Network 32: --- ET01
   RUNG wire#powerrail
      Contact( #Reset_Zona_E0 )
      wire#w1
      Contact( "DB841_Recepcion".DispoArmario[#NumDispo].Protocolo.Reset )
      wire#w2
      S_SR(operand := #Reset_Zona_E1, r1 := wire#w3)
   END_RUNG
   RUNG wire#w1
      Contact( #ZonaUP.Estado.PerReset_CBx )
   END_RUNG wire#w2
   RUNG wire#powerrail
      Contact( #Reset_Zona_E2 )
   END_RUNG wire#w3
   RUNG wire#powerrail
      Contact( #Reset_Zona_E5 )
   END_RUNG wire#w3
   RUNG wire#powerrail
      Contact( #FlancoReset )
   END_RUNG wire#w3
   // the same network as SCL:
   IF #Reset_Zona_E0 AND ("DB841_Recepcion".DispoArmario[#NumDispo].Protocolo.Reset OR #ZonaUP.Estado.PerReset_CBx) THEN
       #Reset_Zona_E1 := TRUE;   // SR flip-flop
   END_IF;
   IF #Reset_Zona_E2 OR #Reset_Zona_E5 OR #FlancoReset THEN #Reset_Zona_E1 := FALSE; END_IF;
END_REGION

REGION Network 33: --- ET00
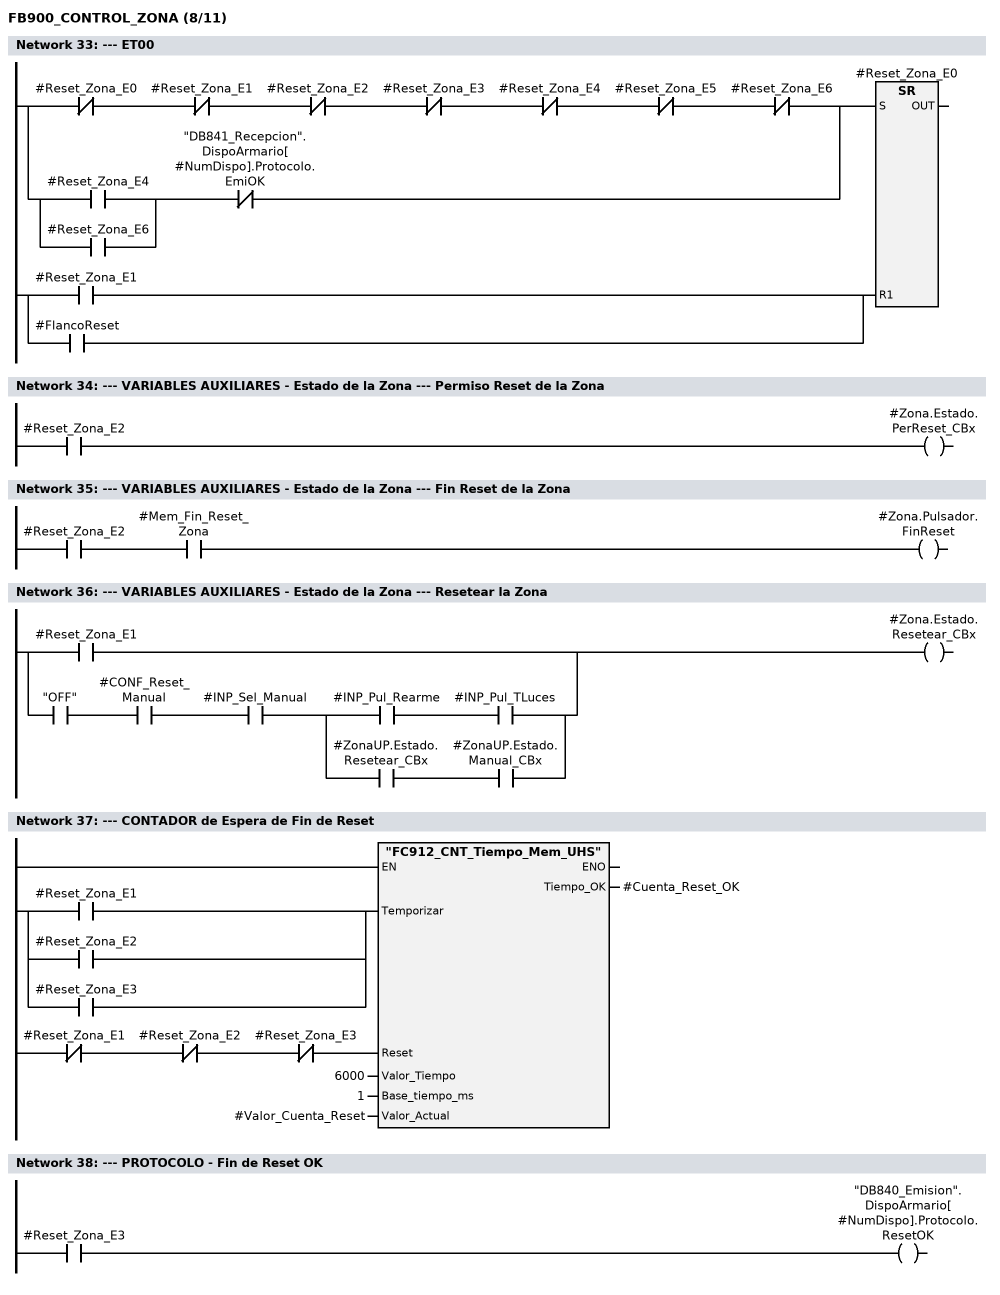
   RUNG wire#powerrail
      I_Contact( #Reset_Zona_E0 )
      I_Contact( #Reset_Zona_E1 )
      I_Contact( #Reset_Zona_E2 )
      I_Contact( #Reset_Zona_E3 )
      I_Contact( #Reset_Zona_E4 )
      I_Contact( #Reset_Zona_E5 )
      I_Contact( #Reset_Zona_E6 )
      wire#w1
      S_SR(operand := #Reset_Zona_E0, r1 := wire#w3)
   END_RUNG
   RUNG wire#powerrail
      Contact( #Reset_Zona_E4 )
      wire#w2
      I_Contact( "DB841_Recepcion".DispoArmario[#NumDispo].Protocolo.EmiOK )
   END_RUNG wire#w1
   RUNG wire#powerrail
      Contact( #Reset_Zona_E6 )
   END_RUNG wire#w2
   RUNG wire#powerrail
      Contact( #Reset_Zona_E1 )
   END_RUNG wire#w3
   RUNG wire#powerrail
      Contact( #FlancoReset )
   END_RUNG wire#w3
   // the same network as SCL:
   IF (NOT #Reset_Zona_E0 AND NOT #Reset_Zona_E1 AND NOT #Reset_Zona_E2 AND NOT #Reset_Zona_E3 AND NOT #Reset_Zona_E4 AND NOT #Reset_Zona_E5 AND NOT #Reset_Zona_E6) OR ((#Reset_Zona_E4 OR #Reset_Zona_E6) AND NOT "DB841_Recepcion".DispoArmario[#NumDispo].Protocolo.EmiOK) THEN
       #Reset_Zona_E0 := TRUE;   // SR flip-flop
   END_IF;
   IF #Reset_Zona_E1 OR #FlancoReset THEN #Reset_Zona_E0 := FALSE; END_IF;
END_REGION

REGION Network 34: --- VARIABLES AUXILIARES - Estado de la Zona --- Permiso Reset de la Zona
   RUNG wire#powerrail
      Contact( #Reset_Zona_E2 )
      Coil( #Zona.Estado.PerReset_CBx )
   END_RUNG
   // the same network as SCL:
   #Zona.Estado.PerReset_CBx := #Reset_Zona_E2;
END_REGION

REGION Network 35: --- VARIABLES AUXILIARES - Estado de la Zona --- Fin Reset de la Zona
   RUNG wire#powerrail
      Contact( #Reset_Zona_E2 )
      Contact( #Mem_Fin_Reset_Zona )
      Coil( #Zona.Pulsador.FinReset )
   END_RUNG
   // the same network as SCL:
   #Zona.Pulsador.FinReset := #Reset_Zona_E2 AND #Mem_Fin_Reset_Zona;
END_REGION

REGION Network 36: --- VARIABLES AUXILIARES - Estado de la Zona --- Resetear la Zona
   RUNG wire#powerrail
      Contact( #Reset_Zona_E1 )
      wire#w1
      Coil( #Zona.Estado.Resetear_CBx )
   END_RUNG
   RUNG wire#powerrail
      Contact( "OFF" )
      Contact( #CONF_Reset_Manual )
      Contact( #INP_Sel_Manual )
      wire#w2
      Contact( #INP_Pul_Rearme )
      Contact( #INP_Pul_TLuces )
   END_RUNG wire#w1
   RUNG wire#w2
      Contact( #ZonaUP.Estado.Resetear_CBx )
      Contact( #ZonaUP.Estado.Manual_CBx )
   END_RUNG wire#w1
   // the same network as SCL:
   #Zona.Estado.Resetear_CBx := #Reset_Zona_E1 OR ("OFF" AND #CONF_Reset_Manual AND #INP_Sel_Manual AND ((#INP_Pul_Rearme AND #INP_Pul_TLuces) OR (#ZonaUP.Estado.Resetear_CBx AND #ZonaUP.Estado.Manual_CBx)));
END_REGION

REGION Network 37: --- CONTADOR de Espera de Fin de Reset
   RUNG wire#powerrail
      "FC912_CNT_Tiempo_Mem_UHS"(Temporizar := wire#w1, Reset := wire#w2, Valor_Tiempo := 6000, Base_tiempo_ms := 1, Valor_Actual := #Valor_Cuenta_Reset, Tiempo_OK => #Cuenta_Reset_OK)
   END_RUNG
   RUNG wire#powerrail
      Contact( #Reset_Zona_E1 )
   END_RUNG wire#w1
   RUNG wire#powerrail
      Contact( #Reset_Zona_E2 )
   END_RUNG wire#w1
   RUNG wire#powerrail
      Contact( #Reset_Zona_E3 )
   END_RUNG wire#w1
   RUNG wire#powerrail
      I_Contact( #Reset_Zona_E1 )
      I_Contact( #Reset_Zona_E2 )
      I_Contact( #Reset_Zona_E3 )
   END_RUNG wire#w2
   // the same network as SCL:
   "FC912_CNT_Tiempo_Mem_UHS"(Temporizar := #Reset_Zona_E1 OR #Reset_Zona_E2 OR #Reset_Zona_E3,
                           Reset := NOT #Reset_Zona_E1 AND NOT #Reset_Zona_E2 AND NOT #Reset_Zona_E3,
                           Valor_Tiempo := 6000,
                           Base_tiempo_ms := 1,
                           Valor_Actual := #Valor_Cuenta_Reset,
                           Tiempo_OK => #Cuenta_Reset_OK);
END_REGION

REGION Network 38: --- PROTOCOLO - Fin de Reset OK
   RUNG wire#powerrail
      Contact( #Reset_Zona_E3 )
      Coil( "DB840_Emision".DispoArmario[#NumDispo].Protocolo.ResetOK )
   END_RUNG
   // the same network as SCL:
   "DB840_Emision".DispoArmario[#NumDispo].Protocolo.ResetOK := #Reset_Zona_E3;
END_REGION

REGION Network 39: --- PROTOCOLO - Fin de Reset No OK
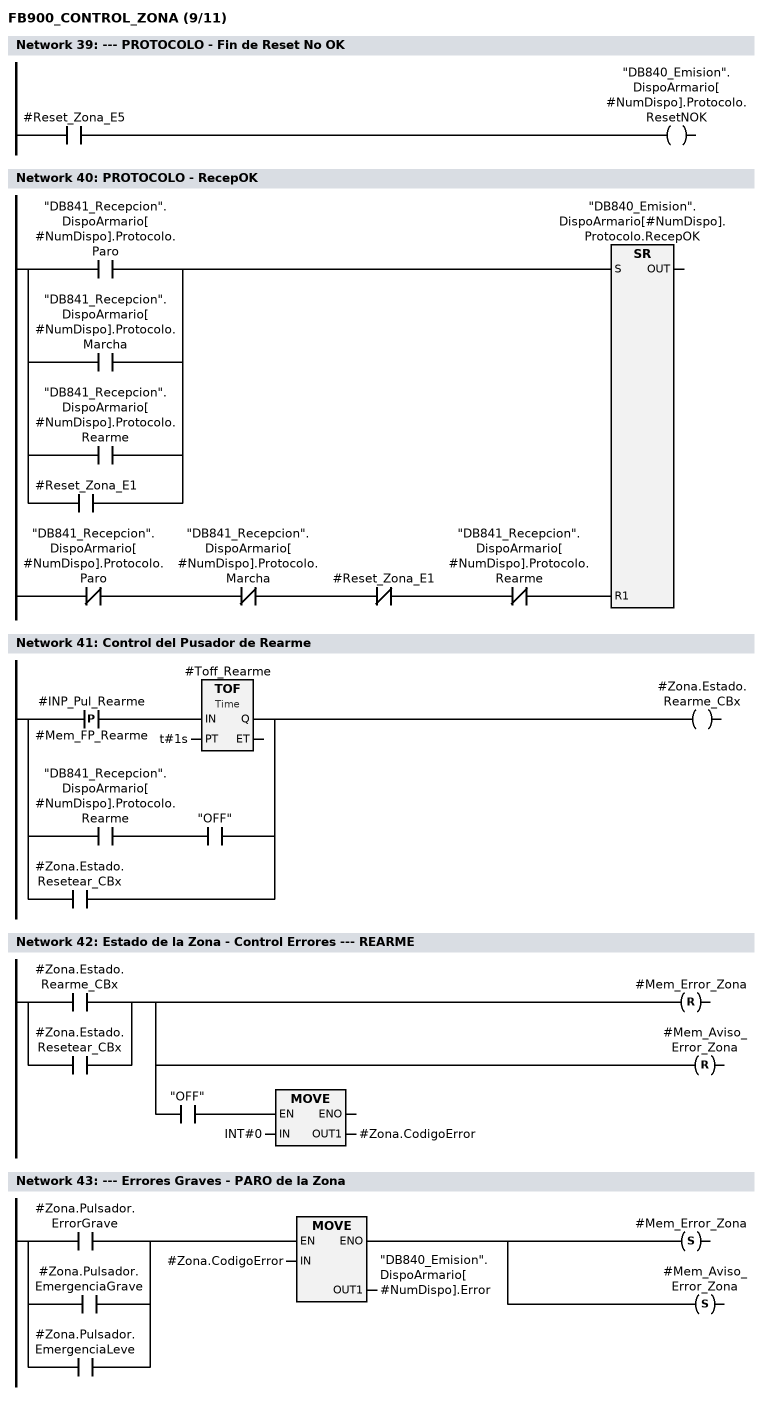
   RUNG wire#powerrail
      Contact( #Reset_Zona_E5 )
      Coil( "DB840_Emision".DispoArmario[#NumDispo].Protocolo.ResetNOK )
   END_RUNG
   // the same network as SCL:
   "DB840_Emision".DispoArmario[#NumDispo].Protocolo.ResetNOK := #Reset_Zona_E5;
END_REGION

REGION Network 40: PROTOCOLO - RecepOK
   RUNG wire#powerrail
      Contact( "DB841_Recepcion".DispoArmario[#NumDispo].Protocolo.Paro )
      wire#w1
      S_SR(operand := "DB840_Emision".DispoArmario[#NumDispo].Protocolo.RecepOK, r1 := wire#w2)
   END_RUNG
   RUNG wire#powerrail
      Contact( "DB841_Recepcion".DispoArmario[#NumDispo].Protocolo.Marcha )
   END_RUNG wire#w1
   RUNG wire#powerrail
      Contact( "DB841_Recepcion".DispoArmario[#NumDispo].Protocolo.Rearme )
   END_RUNG wire#w1
   RUNG wire#powerrail
      Contact( #Reset_Zona_E1 )
   END_RUNG wire#w1
   RUNG wire#powerrail
      I_Contact( "DB841_Recepcion".DispoArmario[#NumDispo].Protocolo.Paro )
      I_Contact( "DB841_Recepcion".DispoArmario[#NumDispo].Protocolo.Marcha )
      I_Contact( #Reset_Zona_E1 )
      I_Contact( "DB841_Recepcion".DispoArmario[#NumDispo].Protocolo.Rearme )
   END_RUNG wire#w2
   // the same network as SCL:
   #_w1 := NOT "DB841_Recepcion".DispoArmario[#NumDispo].Protocolo.Paro AND NOT "DB841_Recepcion".DispoArmario[#NumDispo].Protocolo.Marcha AND NOT #Reset_Zona_E1 AND NOT "DB841_Recepcion".DispoArmario[#NumDispo].Protocolo.Rearme;
   IF "DB841_Recepcion".DispoArmario[#NumDispo].Protocolo.Paro OR "DB841_Recepcion".DispoArmario[#NumDispo].Protocolo.Marcha OR "DB841_Recepcion".DispoArmario[#NumDispo].Protocolo.Rearme OR #Reset_Zona_E1 THEN
       "DB840_Emision".DispoArmario[#NumDispo].Protocolo.RecepOK := TRUE;   // SR flip-flop
   END_IF;
   IF #_w1 THEN "DB840_Emision".DispoArmario[#NumDispo].Protocolo.RecepOK := FALSE; END_IF;
END_REGION

REGION Network 41: Control del Pusador de Rearme
   RUNG wire#powerrail
      P_Contact(operand := #INP_Pul_Rearme, bit := #Mem_FP_Rearme)
      { S7_Templates := "time_type := Time" } #Toff_Rearme.TOF(pt := t#1s, et =>)
      wire#w1
      Coil( #Zona.Estado.Rearme_CBx )
   END_RUNG
   RUNG wire#powerrail
      Contact( "DB841_Recepcion".DispoArmario[#NumDispo].Protocolo.Rearme )
      Contact( "OFF" )
   END_RUNG wire#w1
   RUNG wire#powerrail
      Contact( #Zona.Estado.Resetear_CBx )
   END_RUNG wire#w1
   // the same network as SCL:
   #_w1 := #INP_Pul_Rearme AND NOT #Mem_FP_Rearme;   // rising edge of #INP_Pul_Rearme
   #Mem_FP_Rearme := #INP_Pul_Rearme;
   #Toff_Rearme(IN := #_w1, PT := t#1s);   // TOF
   #Zona.Estado.Rearme_CBx := #Toff_Rearme.Q OR ("DB841_Recepcion".DispoArmario[#NumDispo].Protocolo.Rearme AND "OFF") OR #Zona.Estado.Resetear_CBx;
END_REGION

REGION Network 42: Estado de la Zona - Control Errores --- REARME
   RUNG wire#powerrail
      Contact( #Zona.Estado.Rearme_CBx )
      wire#w1
      R_Coil( #Mem_Error_Zona )
   END_RUNG
   RUNG wire#powerrail
      Contact( #Zona.Estado.Resetear_CBx )
   END_RUNG wire#w1
   RUNG wire#w1
      R_Coil( #Mem_Aviso_Error_Zona )
   END_RUNG
   RUNG wire#w1
      Contact( "OFF" )
      { S7_GenerateENO := "TRUE" } Move(in := INT#0, out1 => #Zona.CodigoError)
   END_RUNG
   // the same network as SCL:
   #_w1 := #Zona.Estado.Rearme_CBx OR #Zona.Estado.Resetear_CBx;
   IF #_w1 THEN
       #Mem_Error_Zona := FALSE;
       #Mem_Aviso_Error_Zona := FALSE;
   END_IF;
   IF #_w1 AND "OFF" THEN #Zona.CodigoError := INT#0; END_IF;
END_REGION

REGION Network 43: --- Errores Graves - PARO de la Zona
   RUNG wire#powerrail
      Contact( #Zona.Pulsador.ErrorGrave )
      wire#w1
      { S7_GenerateENO := "TRUE" } Move(in := #Zona.CodigoError, out1 => "DB840_Emision".DispoArmario[#NumDispo].Error)
      wire#w2
      S_Coil( #Mem_Error_Zona )
   END_RUNG
   RUNG wire#powerrail
      Contact( #Zona.Pulsador.EmergenciaGrave )
   END_RUNG wire#w1
   RUNG wire#powerrail
      Contact( #Zona.Pulsador.EmergenciaLeve )
   END_RUNG wire#w1
   RUNG wire#w2
      S_Coil( #Mem_Aviso_Error_Zona )
   END_RUNG
   // the same network as SCL:
   // ENO of a box is taken as its EN; it also drops when the box reports an error
   IF #Zona.Pulsador.ErrorGrave OR #Zona.Pulsador.EmergenciaGrave OR #Zona.Pulsador.EmergenciaLeve THEN
       "DB840_Emision".DispoArmario[#NumDispo].Error := #Zona.CodigoError;
       #Mem_Error_Zona := TRUE;
       #Mem_Aviso_Error_Zona := TRUE;
   END_IF;
END_REGION

REGION Network 44: Revisar error externo de nivel inferior Olocar Primer Digito
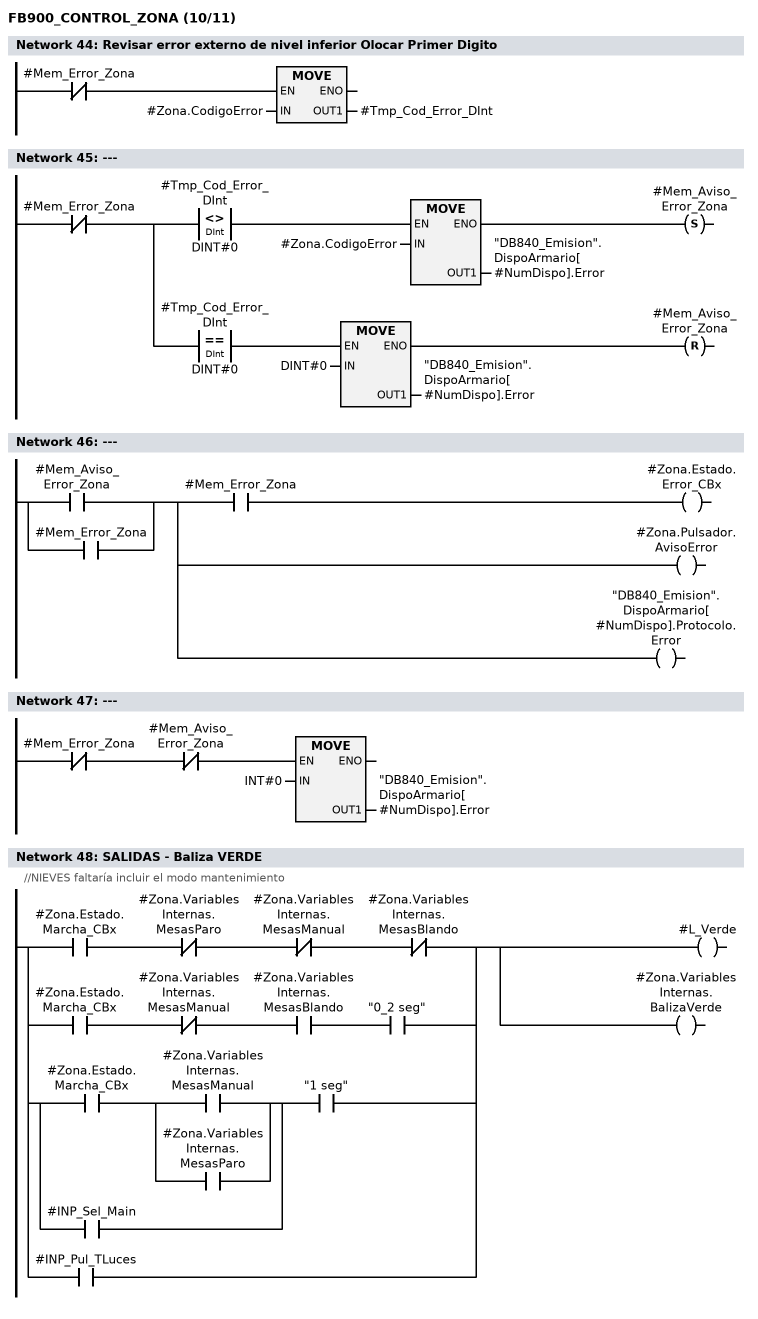
   RUNG wire#powerrail
      I_Contact( #Mem_Error_Zona )
      { S7_GenerateENO := "TRUE" } Move(in := #Zona.CodigoError, out1 => #Tmp_Cod_Error_DInt)
   END_RUNG
   // the same network as SCL:
   IF NOT #Mem_Error_Zona THEN #Tmp_Cod_Error_DInt := #Zona.CodigoError; END_IF;
END_REGION

REGION Network 45: ---
   RUNG wire#powerrail
      I_Contact( #Mem_Error_Zona )
      wire#w1
      { S7_Templates := "SrcType := DInt" } NE_Contact(in1 := #Tmp_Cod_Error_DInt, in2 := DINT#0)
      { S7_GenerateENO := "TRUE" } Move(in := #Zona.CodigoError, out1 => "DB840_Emision".DispoArmario[#NumDispo].Error)
      S_Coil( #Mem_Aviso_Error_Zona )
   END_RUNG
   RUNG wire#w1
      { S7_Templates := "SrcType := DInt" } EQ_Contact(in1 := #Tmp_Cod_Error_DInt, in2 := DINT#0)
      { S7_GenerateENO := "TRUE" } Move(in := DINT#0, out1 => "DB840_Emision".DispoArmario[#NumDispo].Error)
      R_Coil( #Mem_Aviso_Error_Zona )
   END_RUNG
   // the same network as SCL:
   // ENO of a box is taken as its EN; it also drops when the box reports an error
   IF NOT #Mem_Error_Zona AND (#Tmp_Cod_Error_DInt <> DINT#0) THEN
       "DB840_Emision".DispoArmario[#NumDispo].Error := #Zona.CodigoError;
       #Mem_Aviso_Error_Zona := TRUE;
   END_IF;
   IF NOT #Mem_Error_Zona AND (#Tmp_Cod_Error_DInt = DINT#0) THEN
       "DB840_Emision".DispoArmario[#NumDispo].Error := DINT#0;
       #Mem_Aviso_Error_Zona := FALSE;
   END_IF;
END_REGION

REGION Network 46: ---
   RUNG wire#powerrail
      Contact( #Mem_Aviso_Error_Zona )
      wire#w1
      Contact( #Mem_Error_Zona )
      Coil( #Zona.Estado.Error_CBx )
   END_RUNG
   RUNG wire#powerrail
      Contact( #Mem_Error_Zona )
   END_RUNG wire#w1
   RUNG wire#w1
      Coil( #Zona.Pulsador.AvisoError )
   END_RUNG
   RUNG wire#w1
      Coil( "DB840_Emision".DispoArmario[#NumDispo].Protocolo.Error )
   END_RUNG
   // the same network as SCL:
   #_w1 := #Mem_Aviso_Error_Zona OR #Mem_Error_Zona;
   #Zona.Estado.Error_CBx := #_w1 AND #Mem_Error_Zona;
   #Zona.Pulsador.AvisoError := #_w1;
   "DB840_Emision".DispoArmario[#NumDispo].Protocolo.Error := #_w1;
END_REGION

REGION Network 47: ---
   RUNG wire#powerrail
      I_Contact( #Mem_Error_Zona )
      I_Contact( #Mem_Aviso_Error_Zona )
      { S7_GenerateENO := "TRUE" } Move(in := INT#0, out1 => "DB840_Emision".DispoArmario[#NumDispo].Error)
   END_RUNG
   // the same network as SCL:
   IF NOT #Mem_Error_Zona AND NOT #Mem_Aviso_Error_Zona THEN
       "DB840_Emision".DispoArmario[#NumDispo].Error := INT#0;
   END_IF;
END_REGION

REGION Network 48: SALIDAS - Baliza VERDE
   // //NIEVES faltaría incluir el modo mantenimiento
   RUNG wire#powerrail
      Contact( #Zona.Estado.Marcha_CBx )
      I_Contact( #Zona.VariablesInternas.MesasParo )
      I_Contact( #Zona.VariablesInternas.MesasManual )
      I_Contact( #Zona.VariablesInternas.MesasBlando )
      wire#w1
      Coil( #L_Verde )
   END_RUNG
   RUNG wire#powerrail
      Contact( #Zona.Estado.Marcha_CBx )
      I_Contact( #Zona.VariablesInternas.MesasManual )
      Contact( #Zona.VariablesInternas.MesasBlando )
      Contact( "0_2 seg" )
   END_RUNG wire#w1
   RUNG wire#powerrail
      Contact( #Zona.Estado.Marcha_CBx )
      wire#w2
      Contact( #Zona.VariablesInternas.MesasManual )
      wire#w3
      Contact( "1 seg" )
   END_RUNG wire#w1
   RUNG wire#w2
      Contact( #Zona.VariablesInternas.MesasParo )
   END_RUNG wire#w3
   RUNG wire#powerrail
      Contact( #INP_Sel_Main )
   END_RUNG wire#w3
   RUNG wire#powerrail
      Contact( #INP_Pul_TLuces )
   END_RUNG wire#w1
   RUNG wire#w1
      Coil( #Zona.VariablesInternas.BalizaVerde )
   END_RUNG
   // the same network as SCL:
   #L_Verde := (#Zona.Estado.Marcha_CBx AND NOT #Zona.VariablesInternas.MesasParo AND NOT #Zona.VariablesInternas.MesasManual AND NOT #Zona.VariablesInternas.MesasBlando) OR (#Zona.Estado.Marcha_CBx AND NOT #Zona.VariablesInternas.MesasManual AND #Zona.VariablesInternas.MesasBlando AND "0_2 seg") OR (((#Zona.Estado.Marcha_CBx AND (#Zona.VariablesInternas.MesasManual OR #Zona.VariablesInternas.MesasParo)) OR #INP_Sel_Main) AND "1 seg") OR #INP_Pul_TLuces;
   #Zona.VariablesInternas.BalizaVerde := #L_Verde;
END_REGION

REGION Network 49: SALIDAS - Baliza NARANJA
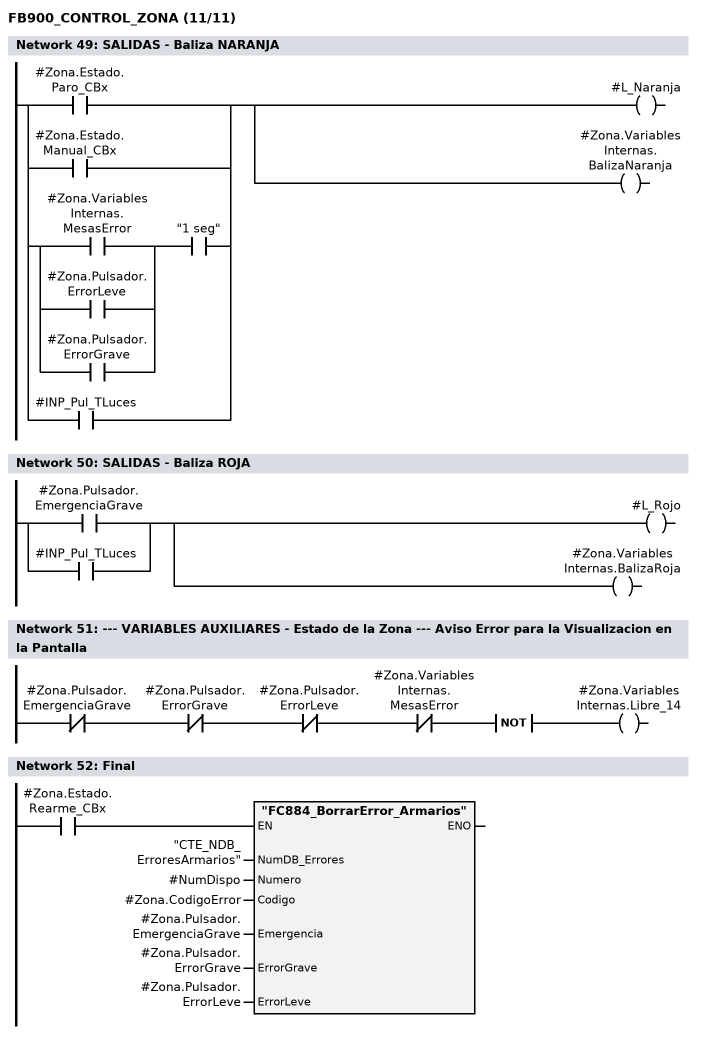
   RUNG wire#powerrail
      Contact( #Zona.Estado.Paro_CBx )
      wire#w1
      Coil( #L_Naranja )
   END_RUNG
   RUNG wire#powerrail
      Contact( #Zona.Estado.Manual_CBx )
   END_RUNG wire#w1
   RUNG wire#powerrail
      Contact( #Zona.VariablesInternas.MesasError )
      wire#w2
      Contact( "1 seg" )
   END_RUNG wire#w1
   RUNG wire#powerrail
      Contact( #Zona.Pulsador.ErrorLeve )
   END_RUNG wire#w2
   RUNG wire#powerrail
      Contact( #Zona.Pulsador.ErrorGrave )
   END_RUNG wire#w2
   RUNG wire#powerrail
      Contact( #INP_Pul_TLuces )
   END_RUNG wire#w1
   RUNG wire#w1
      Coil( #Zona.VariablesInternas.BalizaNaranja )
   END_RUNG
   // the same network as SCL:
   #L_Naranja := #Zona.Estado.Paro_CBx OR #Zona.Estado.Manual_CBx OR ((#Zona.VariablesInternas.MesasError OR #Zona.Pulsador.ErrorLeve OR #Zona.Pulsador.ErrorGrave) AND "1 seg") OR #INP_Pul_TLuces;
   #Zona.VariablesInternas.BalizaNaranja := #L_Naranja;
END_REGION

REGION Network 50: SALIDAS - Baliza ROJA
   RUNG wire#powerrail
      Contact( #Zona.Pulsador.EmergenciaGrave )
      wire#w1
      Coil( #L_Rojo )
   END_RUNG
   RUNG wire#powerrail
      Contact( #INP_Pul_TLuces )
   END_RUNG wire#w1
   RUNG wire#w1
      Coil( #Zona.VariablesInternas.BalizaRoja )
   END_RUNG
   // the same network as SCL:
   #L_Rojo := #Zona.Pulsador.EmergenciaGrave OR #INP_Pul_TLuces;
   #Zona.VariablesInternas.BalizaRoja := #L_Rojo;
END_REGION

REGION Network 51: --- VARIABLES AUXILIARES - Estado de la Zona --- Aviso Error para la Visualizacion en la Pantalla
   RUNG wire#powerrail
      I_Contact( #Zona.Pulsador.EmergenciaGrave )
      I_Contact( #Zona.Pulsador.ErrorGrave )
      I_Contact( #Zona.Pulsador.ErrorLeve )
      I_Contact( #Zona.VariablesInternas.MesasError )
      Not()
      Coil( #Zona.VariablesInternas.Libre_14 )
   END_RUNG
   // the same network as SCL:
   #Zona.VariablesInternas.Libre_14 := NOT (NOT #Zona.Pulsador.EmergenciaGrave AND NOT #Zona.Pulsador.ErrorGrave AND NOT #Zona.Pulsador.ErrorLeve AND NOT #Zona.VariablesInternas.MesasError);
END_REGION

REGION Network 52: Final
   RUNG wire#powerrail
      Contact( #Zona.Estado.Rearme_CBx )
      "FC884_BorrarError_Armarios"(NumDB_Errores := "CTE_NDB_ErroresArmarios", Numero := #NumDispo, Codigo := #Zona.CodigoError, Emergencia := #Zona.Pulsador.EmergenciaGrave, ErrorGrave := #Zona.Pulsador.ErrorGrave, ErrorLeve := #Zona.Pulsador.ErrorLeve)
   END_RUNG
   // the same network as SCL:
   IF #Zona.Estado.Rearme_CBx THEN
       "FC884_BorrarError_Armarios"(NumDB_Errores := "CTE_NDB_ErroresArmarios",
                               Numero := #NumDispo,
                               Codigo := #Zona.CodigoError,
                               Emergencia := #Zona.Pulsador.EmergenciaGrave,
                               ErrorGrave := #Zona.Pulsador.ErrorGrave,
                               ErrorLeve := #Zona.Pulsador.ErrorLeve);
   END_IF;
END_REGION

NETWORK
TITLE = ---
// ---------------------------------------------------------------------
// --- Paso 1 : Escribir datos del DB de Zona

      CALL  BLKMOV
      ( SRCBLK  := #Zona,
        RET_VAL := #ValorReturn,
        DSTBLK  := "DB901_Estado_Zonas".EstadoZona[#NumDispo]
      );


// ---------------------------------------------------------------------
// --- Datos para el Scada

      L     #NumZona;
      T     #NumDispo;

      CALL  "FC962_ScadaZona"
      ( NumZona     := #NumDispo,
        P_Marcha    := #INP_Pul_Marcha,
        P_Paro      := #INP_Pul_Paro,
        P_Rearme    := #INP_Pul_Rearme,
        P_TestLuces := #INP_Pul_TLuces,
        P_Auto      := #INP_Sel_Automat,
        P_OffLine   := #INP_Sel_OffLine,
        P_Main      := #INP_Sel_Main,
        H_Verde     := #Zona.VariablesInternas.BalizaVerde,
        H_Roja      := #Zona.VariablesInternas.BalizaRoja,
        H_Naranja   := #Zona.VariablesInternas.BalizaNaranja
      );


END_FUNCTION_BLOCK
